Omron Sysmac Studio project ethercat (Sysmac Studio 1.23.0.14, StandardProject)

# Controller new_Controller_0: NX1P2-1040DT1 version 1.18
Task PrimaryTask (priority 4, period or condition 8000): Programa0
Library INV00x_MX2_ECT 1.0.9 (contents left out)

VAR_GLOBAL
    PP : BOOL;  (* at BuiltInIO://cpu/#0/Input_Bit_00 *)
    PM : BOOL;  (* at BuiltInIO://cpu/#0/Input_Bit_01 *)
    Variador_01_Comando : WORD;  (* at ECAT://node#11/Command *)
    Variador_01_Frecuencia : UINT;  (* at ECAT://node#11/Frequency reference *)
END_VAR

PROGRAM Programa0
VAR
    Sentido : BOOL;
    Tiempo_1 : BOOL;
    Tiempo_2 : BOOL;
    Trigger_1 : BOOL;
    Trigger_2 : BOOL;
    timer_1_status : _sTimer;
    timer_2_status : _sTimer;
    elapsed_1 : UINT;
    elapsed_2 : UINT;
    Trigger_3 : BOOL;
    timer_3_status : _sTimer;
    Tiempo_3 : BOOL;
    elapsed_3 : UINT;
END_VAR
VAR_EXTERNAL
    PM : BOOL;
    Variador_01_Comando : WORD;
    PP : BOOL;
    Variador_01_Frecuencia : UINT;
END_VAR

(* Section main: ladder, written here as Structured Text *)

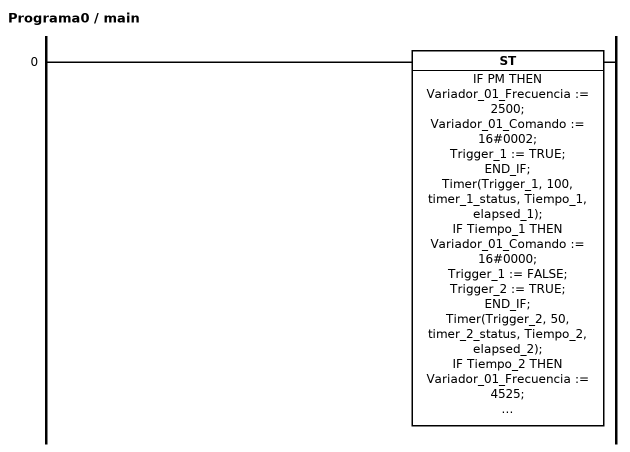
(* Rung 0 *)
IF PM THEN
	Variador_01_Frecuencia := 2500;
	Variador_01_Comando := 16#0002;
	Trigger_1 := TRUE;
END_IF;

Timer(Trigger_1, 100, timer_1_status, Tiempo_1, elapsed_1);

IF Tiempo_1 THEN
	Variador_01_Comando := 16#0000;
	Trigger_1 := FALSE;
	Trigger_2 := TRUE;
END_IF;

Timer(Trigger_2, 50, timer_2_status, Tiempo_2, elapsed_2);

IF Tiempo_2 THEN
	Variador_01_Frecuencia := 4525;
	Variador_01_Comando := 16#0002;
	Trigger_2 := FALSE;
	Trigger_3 := TRUE;
END_IF;

Timer(Trigger_3, 120, timer_3_status, Tiempo_3, elapsed_3);

IF Tiempo_3 THEN
	Variador_01_Comando := 16#0000;
	Trigger_3 := FALSE;
END_IF;
END_PROGRAM